// TIA Portal V17 export
// export: Created 2022-03-12T16:05:29.4048686Z, ExportSetting WithDefaults, DisplayName Totally Integrated Automation Portal, DisplayVersion V17, DisplayName TIA Portal Openness, DisplayVersion V17, DisplayName TIA Portal Version Control Interface, DisplayVersion V17, DisplayName STEP 7 Professional, DisplayVersion V17, DisplayName STEP 7 Safety, DisplayVersion V17, DisplayName WinCC Advanced / Unified PC, DisplayVersion V17
DATA_BLOCK "MessagePrefix"   // DB31604
TITLE = CPG_MessagePrefix
{ S7_Optimized_Access := 'TRUE' }
AUTHOR : tech.team.motioncontrol@siemens.com
FAMILY : CPG
VERSION : 1.0
// Support: tech.team.motioncontrol@siemens.com
// Fax: +49 (0) 9131/98-1297
// stored: AutoNumber true, DBAccessibleFromOPCUA true, DBAccessibleFromWebserver true, IsOnlyStoredInLoadMemory false, IsRetainMemResEnabled false, IsWriteProtectedInAS false, MemoryReserve 0
   VAR
      UN { ExternalAccessible := 'False'; ExternalVisible := 'False'; ExternalWritable := 'False'} : Struct   // MessagePrefix for Unit
         Alarm { ExternalAccessible := 'False'; ExternalVisible := 'False'; ExternalWritable := 'False'; S7_SetPoint := 'True'} : "CPG_typeMessagePrefix";   // MessagePrefix for Unit Alarms
      END_STRUCT;
      EM00 { ExternalAccessible := 'False'; ExternalVisible := 'False'; ExternalWritable := 'False'} : Struct   // MessagePrefix for EquipmentModuleEM00
         EventControl { ExternalAccessible := 'False'; ExternalVisible := 'False'; ExternalWritable := 'False'; S7_SetPoint := 'True'} : "CPG_typeMessagePrefix";   // MessagePrefixforEventControl
         CM01 { ExternalAccessible := 'False'; ExternalVisible := 'False'; ExternalWritable := 'False'; S7_SetPoint := 'True'} : "CPG_typeMessagePrefix";   // MessagePrefixforControlModule#01
         CM02 { ExternalAccessible := 'False'; ExternalVisible := 'False'; ExternalWritable := 'False'; S7_SetPoint := 'True'} : "CPG_typeMessagePrefix";   // MessagePrefixforControlModule#02
         CM03 { ExternalAccessible := 'False'; ExternalVisible := 'False'; ExternalWritable := 'False'; S7_SetPoint := 'True'} : "CPG_typeMessagePrefix";   // MessagePrefixforControlModule#03
         CM04 { ExternalAccessible := 'False'; ExternalVisible := 'False'; ExternalWritable := 'False'; S7_SetPoint := 'True'} : "CPG_typeMessagePrefix";   // MessagePrefixforControlModule#04
         CM05 { ExternalAccessible := 'False'; ExternalVisible := 'False'; ExternalWritable := 'False'; S7_SetPoint := 'True'} : "CPG_typeMessagePrefix";   // MessagePrefixforControlModule#05
         CM06 { ExternalAccessible := 'False'; ExternalVisible := 'False'; ExternalWritable := 'False'; S7_SetPoint := 'True'} : "CPG_typeMessagePrefix";   // MessagePrefixforControlModule#06
         CM07 { ExternalAccessible := 'False'; ExternalVisible := 'False'; ExternalWritable := 'False'; S7_SetPoint := 'True'} : "CPG_typeMessagePrefix";   // MessagePrefixforControlModule#07
         CM08 { ExternalAccessible := 'False'; ExternalVisible := 'False'; ExternalWritable := 'False'; S7_SetPoint := 'True'} : "CPG_typeMessagePrefix";   // MessagePrefixforControlModule#08
         CM09 { ExternalAccessible := 'False'; ExternalVisible := 'False'; ExternalWritable := 'False'; S7_SetPoint := 'True'} : "CPG_typeMessagePrefix";   // MessagePrefixforControlModule#09
         CM10 { ExternalAccessible := 'False'; ExternalVisible := 'False'; ExternalWritable := 'False'; S7_SetPoint := 'True'} : "CPG_typeMessagePrefix";   // MessagePrefixforControlModule#10
      END_STRUCT;
      EM01 { ExternalAccessible := 'False'; ExternalVisible := 'False'; ExternalWritable := 'False'} : Struct   // MessagePrefix for EquipmentModuleEM01
         EventControl { ExternalAccessible := 'False'; ExternalVisible := 'False'; ExternalWritable := 'False'; S7_SetPoint := 'True'} : "CPG_typeMessagePrefix";   // MessagePrefixforEventControl
         CM01 { ExternalAccessible := 'False'; ExternalVisible := 'False'; ExternalWritable := 'False'; S7_SetPoint := 'True'} : "CPG_typeMessagePrefix";   // MessagePrefixforControlModule#01
         CM02 { ExternalAccessible := 'False'; ExternalVisible := 'False'; ExternalWritable := 'False'; S7_SetPoint := 'True'} : "CPG_typeMessagePrefix";   // MessagePrefixforControlModule#02
         CM03 { ExternalAccessible := 'False'; ExternalVisible := 'False'; ExternalWritable := 'False'; S7_SetPoint := 'True'} : "CPG_typeMessagePrefix";   // MessagePrefixforControlModule#03
         CM04 { ExternalAccessible := 'False'; ExternalVisible := 'False'; ExternalWritable := 'False'; S7_SetPoint := 'True'} : "CPG_typeMessagePrefix";   // MessagePrefixforControlModule#04
         CM05 { ExternalAccessible := 'False'; ExternalVisible := 'False'; ExternalWritable := 'False'; S7_SetPoint := 'True'} : "CPG_typeMessagePrefix";   // MessagePrefixforControlModule#05
         CM06 { ExternalAccessible := 'False'; ExternalVisible := 'False'; ExternalWritable := 'False'; S7_SetPoint := 'True'} : "CPG_typeMessagePrefix";   // MessagePrefixforControlModule#06
         CM07 { ExternalAccessible := 'False'; ExternalVisible := 'False'; ExternalWritable := 'False'; S7_SetPoint := 'True'} : "CPG_typeMessagePrefix";   // MessagePrefixforControlModule#07
         CM08 { ExternalAccessible := 'False'; ExternalVisible := 'False'; ExternalWritable := 'False'; S7_SetPoint := 'True'} : "CPG_typeMessagePrefix";   // MessagePrefixforControlModule#08
         CM09 { ExternalAccessible := 'False'; ExternalVisible := 'False'; ExternalWritable := 'False'; S7_SetPoint := 'True'} : "CPG_typeMessagePrefix";   // MessagePrefixforControlModule#09
         CM10 { ExternalAccessible := 'False'; ExternalVisible := 'False'; ExternalWritable := 'False'; S7_SetPoint := 'True'} : "CPG_typeMessagePrefix";   // MessagePrefixforControlModule#10
      END_STRUCT;
      EM02 { ExternalAccessible := 'False'; ExternalVisible := 'False'; ExternalWritable := 'False'} : Struct   // MessagePrefix for EquipmentModuleEM02
         EventControl { ExternalAccessible := 'False'; ExternalVisible := 'False'; ExternalWritable := 'False'; S7_SetPoint := 'True'} : "CPG_typeMessagePrefix";   // MessagePrefixforEventControl
         CM01 { ExternalAccessible := 'False'; ExternalVisible := 'False'; ExternalWritable := 'False'; S7_SetPoint := 'True'} : "CPG_typeMessagePrefix";   // MessagePrefixforControlModule#01
         CM02 { ExternalAccessible := 'False'; ExternalVisible := 'False'; ExternalWritable := 'False'; S7_SetPoint := 'True'} : "CPG_typeMessagePrefix";   // MessagePrefixforControlModule#02
         CM03 { ExternalAccessible := 'False'; ExternalVisible := 'False'; ExternalWritable := 'False'; S7_SetPoint := 'True'} : "CPG_typeMessagePrefix";   // MessagePrefixforControlModule#03
         CM04 { ExternalAccessible := 'False'; ExternalVisible := 'False'; ExternalWritable := 'False'; S7_SetPoint := 'True'} : "CPG_typeMessagePrefix";   // MessagePrefixforControlModule#04
         CM05 { ExternalAccessible := 'False'; ExternalVisible := 'False'; ExternalWritable := 'False'; S7_SetPoint := 'True'} : "CPG_typeMessagePrefix";   // MessagePrefixforControlModule#05
         CM06 { ExternalAccessible := 'False'; ExternalVisible := 'False'; ExternalWritable := 'False'; S7_SetPoint := 'True'} : "CPG_typeMessagePrefix";   // MessagePrefixforControlModule#06
         CM07 { ExternalAccessible := 'False'; ExternalVisible := 'False'; ExternalWritable := 'False'; S7_SetPoint := 'True'} : "CPG_typeMessagePrefix";   // MessagePrefixforControlModule#07
         CM08 { ExternalAccessible := 'False'; ExternalVisible := 'False'; ExternalWritable := 'False'; S7_SetPoint := 'True'} : "CPG_typeMessagePrefix";   // MessagePrefixforControlModule#08
         CM09 { ExternalAccessible := 'False'; ExternalVisible := 'False'; ExternalWritable := 'False'; S7_SetPoint := 'True'} : "CPG_typeMessagePrefix";   // MessagePrefixforControlModule#09
         CM10 { ExternalAccessible := 'False'; ExternalVisible := 'False'; ExternalWritable := 'False'; S7_SetPoint := 'True'} : "CPG_typeMessagePrefix";   // MessagePrefixforControlModule#10
      END_STRUCT;
      EM03 { ExternalAccessible := 'False'; ExternalVisible := 'False'; ExternalWritable := 'False'} : Struct   // MessagePrefix for EquipmentModuleEM03
         EventControl { ExternalAccessible := 'False'; ExternalVisible := 'False'; ExternalWritable := 'False'; S7_SetPoint := 'True'} : "CPG_typeMessagePrefix";   // MessagePrefixforEventControl
         CM01 { ExternalAccessible := 'False'; ExternalVisible := 'False'; ExternalWritable := 'False'; S7_SetPoint := 'True'} : "CPG_typeMessagePrefix";   // MessagePrefixforControlModule#01
         CM02 { ExternalAccessible := 'False'; ExternalVisible := 'False'; ExternalWritable := 'False'; S7_SetPoint := 'True'} : "CPG_typeMessagePrefix";   // MessagePrefixforControlModule#02
         CM03 { ExternalAccessible := 'False'; ExternalVisible := 'False'; ExternalWritable := 'False'; S7_SetPoint := 'True'} : "CPG_typeMessagePrefix";   // MessagePrefixforControlModule#03
         CM04 { ExternalAccessible := 'False'; ExternalVisible := 'False'; ExternalWritable := 'False'; S7_SetPoint := 'True'} : "CPG_typeMessagePrefix";   // MessagePrefixforControlModule#04
         CM05 { ExternalAccessible := 'False'; ExternalVisible := 'False'; ExternalWritable := 'False'; S7_SetPoint := 'True'} : "CPG_typeMessagePrefix";   // MessagePrefixforControlModule#05
         CM06 { ExternalAccessible := 'False'; ExternalVisible := 'False'; ExternalWritable := 'False'; S7_SetPoint := 'True'} : "CPG_typeMessagePrefix";   // MessagePrefixforControlModule#06
         CM07 { ExternalAccessible := 'False'; ExternalVisible := 'False'; ExternalWritable := 'False'; S7_SetPoint := 'True'} : "CPG_typeMessagePrefix";   // MessagePrefixforControlModule#07
         CM08 { ExternalAccessible := 'False'; ExternalVisible := 'False'; ExternalWritable := 'False'; S7_SetPoint := 'True'} : "CPG_typeMessagePrefix";   // MessagePrefixforControlModule#08
         CM09 { ExternalAccessible := 'False'; ExternalVisible := 'False'; ExternalWritable := 'False'; S7_SetPoint := 'True'} : "CPG_typeMessagePrefix";   // MessagePrefixforControlModule#09
         CM10 { ExternalAccessible := 'False'; ExternalVisible := 'False'; ExternalWritable := 'False'; S7_SetPoint := 'True'} : "CPG_typeMessagePrefix";   // MessagePrefixforControlModule#10
      END_STRUCT;
      EM04 { ExternalAccessible := 'False'; ExternalVisible := 'False'; ExternalWritable := 'False'} : Struct   // MessagePrefix for EquipmentModuleEM04
         EventControl { ExternalAccessible := 'False'; ExternalVisible := 'False'; ExternalWritable := 'False'; S7_SetPoint := 'True'} : "CPG_typeMessagePrefix";   // MessagePrefixforEventControl
         CM01 { ExternalAccessible := 'False'; ExternalVisible := 'False'; ExternalWritable := 'False'; S7_SetPoint := 'True'} : "CPG_typeMessagePrefix";   // MessagePrefixforControlModule#01
         CM02 { ExternalAccessible := 'False'; ExternalVisible := 'False'; ExternalWritable := 'False'; S7_SetPoint := 'True'} : "CPG_typeMessagePrefix";   // MessagePrefixforControlModule#02
         CM03 { ExternalAccessible := 'False'; ExternalVisible := 'False'; ExternalWritable := 'False'; S7_SetPoint := 'True'} : "CPG_typeMessagePrefix";   // MessagePrefixforControlModule#03
         CM04 { ExternalAccessible := 'False'; ExternalVisible := 'False'; ExternalWritable := 'False'; S7_SetPoint := 'True'} : "CPG_typeMessagePrefix";   // MessagePrefixforControlModule#04
         CM05 { ExternalAccessible := 'False'; ExternalVisible := 'False'; ExternalWritable := 'False'; S7_SetPoint := 'True'} : "CPG_typeMessagePrefix";   // MessagePrefixforControlModule#05
         CM06 { ExternalAccessible := 'False'; ExternalVisible := 'False'; ExternalWritable := 'False'; S7_SetPoint := 'True'} : "CPG_typeMessagePrefix";   // MessagePrefixforControlModule#06
         CM07 { ExternalAccessible := 'False'; ExternalVisible := 'False'; ExternalWritable := 'False'; S7_SetPoint := 'True'} : "CPG_typeMessagePrefix";   // MessagePrefixforControlModule#07
         CM08 { ExternalAccessible := 'False'; ExternalVisible := 'False'; ExternalWritable := 'False'; S7_SetPoint := 'True'} : "CPG_typeMessagePrefix";   // MessagePrefixforControlModule#08
         CM09 { ExternalAccessible := 'False'; ExternalVisible := 'False'; ExternalWritable := 'False'; S7_SetPoint := 'True'} : "CPG_typeMessagePrefix";   // MessagePrefixforControlModule#09
         CM10 { ExternalAccessible := 'False'; ExternalVisible := 'False'; ExternalWritable := 'False'; S7_SetPoint := 'True'} : "CPG_typeMessagePrefix";   // MessagePrefixforControlModule#10
      END_STRUCT;
      EM05 { ExternalAccessible := 'False'; ExternalVisible := 'False'; ExternalWritable := 'False'} : Struct   // MessagePrefix for EquipmentModuleEM05
         EventControl { ExternalAccessible := 'False'; ExternalVisible := 'False'; ExternalWritable := 'False'; S7_SetPoint := 'True'} : "CPG_typeMessagePrefix";   // MessagePrefixforEventControl
         CM01 { ExternalAccessible := 'False'; ExternalVisible := 'False'; ExternalWritable := 'False'; S7_SetPoint := 'True'} : "CPG_typeMessagePrefix";   // MessagePrefixforControlModule#01
         CM02 { ExternalAccessible := 'False'; ExternalVisible := 'False'; ExternalWritable := 'False'; S7_SetPoint := 'True'} : "CPG_typeMessagePrefix";   // MessagePrefixforControlModule#02
         CM03 { ExternalAccessible := 'False'; ExternalVisible := 'False'; ExternalWritable := 'False'; S7_SetPoint := 'True'} : "CPG_typeMessagePrefix";   // MessagePrefixforControlModule#03
         CM04 { ExternalAccessible := 'False'; ExternalVisible := 'False'; ExternalWritable := 'False'; S7_SetPoint := 'True'} : "CPG_typeMessagePrefix";   // MessagePrefixforControlModule#04
         CM05 { ExternalAccessible := 'False'; ExternalVisible := 'False'; ExternalWritable := 'False'; S7_SetPoint := 'True'} : "CPG_typeMessagePrefix";   // MessagePrefixforControlModule#05
         CM06 { ExternalAccessible := 'False'; ExternalVisible := 'False'; ExternalWritable := 'False'; S7_SetPoint := 'True'} : "CPG_typeMessagePrefix";   // MessagePrefixforControlModule#06
         CM07 { ExternalAccessible := 'False'; ExternalVisible := 'False'; ExternalWritable := 'False'; S7_SetPoint := 'True'} : "CPG_typeMessagePrefix";   // MessagePrefixforControlModule#07
         CM08 { ExternalAccessible := 'False'; ExternalVisible := 'False'; ExternalWritable := 'False'; S7_SetPoint := 'True'} : "CPG_typeMessagePrefix";   // MessagePrefixforControlModule#08
         CM09 { ExternalAccessible := 'False'; ExternalVisible := 'False'; ExternalWritable := 'False'; S7_SetPoint := 'True'} : "CPG_typeMessagePrefix";   // MessagePrefixforControlModule#09
         CM10 { ExternalAccessible := 'False'; ExternalVisible := 'False'; ExternalWritable := 'False'; S7_SetPoint := 'True'} : "CPG_typeMessagePrefix";   // MessagePrefixforControlModule#10
      END_STRUCT;
      EM06 { ExternalAccessible := 'False'; ExternalVisible := 'False'; ExternalWritable := 'False'} : Struct   // MessagePrefix for EquipmentModuleEM06
         EventControl { ExternalAccessible := 'False'; ExternalVisible := 'False'; ExternalWritable := 'False'; S7_SetPoint := 'True'} : "CPG_typeMessagePrefix";   // MessagePrefixforEventControl
         CM01 { ExternalAccessible := 'False'; ExternalVisible := 'False'; ExternalWritable := 'False'; S7_SetPoint := 'True'} : "CPG_typeMessagePrefix";   // MessagePrefixforControlModule#01
         CM02 { ExternalAccessible := 'False'; ExternalVisible := 'False'; ExternalWritable := 'False'; S7_SetPoint := 'True'} : "CPG_typeMessagePrefix";   // MessagePrefixforControlModule#02
         CM03 { ExternalAccessible := 'False'; ExternalVisible := 'False'; ExternalWritable := 'False'; S7_SetPoint := 'True'} : "CPG_typeMessagePrefix";   // MessagePrefixforControlModule#03
         CM04 { ExternalAccessible := 'False'; ExternalVisible := 'False'; ExternalWritable := 'False'; S7_SetPoint := 'True'} : "CPG_typeMessagePrefix";   // MessagePrefixforControlModule#04
         CM05 { ExternalAccessible := 'False'; ExternalVisible := 'False'; ExternalWritable := 'False'; S7_SetPoint := 'True'} : "CPG_typeMessagePrefix";   // MessagePrefixforControlModule#05
         CM06 { ExternalAccessible := 'False'; ExternalVisible := 'False'; ExternalWritable := 'False'; S7_SetPoint := 'True'} : "CPG_typeMessagePrefix";   // MessagePrefixforControlModule#06
         CM07 { ExternalAccessible := 'False'; ExternalVisible := 'False'; ExternalWritable := 'False'; S7_SetPoint := 'True'} : "CPG_typeMessagePrefix";   // MessagePrefixforControlModule#07
         CM08 { ExternalAccessible := 'False'; ExternalVisible := 'False'; ExternalWritable := 'False'; S7_SetPoint := 'True'} : "CPG_typeMessagePrefix";   // MessagePrefixforControlModule#08
         CM09 { ExternalAccessible := 'False'; ExternalVisible := 'False'; ExternalWritable := 'False'; S7_SetPoint := 'True'} : "CPG_typeMessagePrefix";   // MessagePrefixforControlModule#09
         CM10 { ExternalAccessible := 'False'; ExternalVisible := 'False'; ExternalWritable := 'False'; S7_SetPoint := 'True'} : "CPG_typeMessagePrefix";   // MessagePrefixforControlModule#10
      END_STRUCT;
      EM07 { ExternalAccessible := 'False'; ExternalVisible := 'False'; ExternalWritable := 'False'} : Struct   // MessagePrefix for EquipmentModuleEM07
         EventControl { ExternalAccessible := 'False'; ExternalVisible := 'False'; ExternalWritable := 'False'; S7_SetPoint := 'True'} : "CPG_typeMessagePrefix";   // MessagePrefixforEventControl
         CM01 { ExternalAccessible := 'False'; ExternalVisible := 'False'; ExternalWritable := 'False'; S7_SetPoint := 'True'} : "CPG_typeMessagePrefix";   // MessagePrefixforControlModule#01
         CM02 { ExternalAccessible := 'False'; ExternalVisible := 'False'; ExternalWritable := 'False'; S7_SetPoint := 'True'} : "CPG_typeMessagePrefix";   // MessagePrefixforControlModule#02
         CM03 { ExternalAccessible := 'False'; ExternalVisible := 'False'; ExternalWritable := 'False'; S7_SetPoint := 'True'} : "CPG_typeMessagePrefix";   // MessagePrefixforControlModule#03
         CM04 { ExternalAccessible := 'False'; ExternalVisible := 'False'; ExternalWritable := 'False'; S7_SetPoint := 'True'} : "CPG_typeMessagePrefix";   // MessagePrefixforControlModule#04
         CM05 { ExternalAccessible := 'False'; ExternalVisible := 'False'; ExternalWritable := 'False'; S7_SetPoint := 'True'} : "CPG_typeMessagePrefix";   // MessagePrefixforControlModule#05
         CM06 { ExternalAccessible := 'False'; ExternalVisible := 'False'; ExternalWritable := 'False'; S7_SetPoint := 'True'} : "CPG_typeMessagePrefix";   // MessagePrefixforControlModule#06
         CM07 { ExternalAccessible := 'False'; ExternalVisible := 'False'; ExternalWritable := 'False'; S7_SetPoint := 'True'} : "CPG_typeMessagePrefix";   // MessagePrefixforControlModule#07
         CM08 { ExternalAccessible := 'False'; ExternalVisible := 'False'; ExternalWritable := 'False'; S7_SetPoint := 'True'} : "CPG_typeMessagePrefix";   // MessagePrefixforControlModule#08
         CM09 { ExternalAccessible := 'False'; ExternalVisible := 'False'; ExternalWritable := 'False'; S7_SetPoint := 'True'} : "CPG_typeMessagePrefix";   // MessagePrefixforControlModule#09
         CM10 { ExternalAccessible := 'False'; ExternalVisible := 'False'; ExternalWritable := 'False'; S7_SetPoint := 'True'} : "CPG_typeMessagePrefix";   // MessagePrefixforControlModule#10
      END_STRUCT;
      EM08 { ExternalAccessible := 'False'; ExternalVisible := 'False'; ExternalWritable := 'False'} : Struct   // MessagePrefix for EquipmentModuleEM08
         EventControl { ExternalAccessible := 'False'; ExternalVisible := 'False'; ExternalWritable := 'False'; S7_SetPoint := 'True'} : "CPG_typeMessagePrefix";   // MessagePrefixforEventControl
         CM01 { ExternalAccessible := 'False'; ExternalVisible := 'False'; ExternalWritable := 'False'; S7_SetPoint := 'True'} : "CPG_typeMessagePrefix";   // MessagePrefixforControlModule#01
         CM02 { ExternalAccessible := 'False'; ExternalVisible := 'False'; ExternalWritable := 'False'; S7_SetPoint := 'True'} : "CPG_typeMessagePrefix";   // MessagePrefixforControlModule#02
         CM03 { ExternalAccessible := 'False'; ExternalVisible := 'False'; ExternalWritable := 'False'; S7_SetPoint := 'True'} : "CPG_typeMessagePrefix";   // MessagePrefixforControlModule#03
         CM04 { ExternalAccessible := 'False'; ExternalVisible := 'False'; ExternalWritable := 'False'; S7_SetPoint := 'True'} : "CPG_typeMessagePrefix";   // MessagePrefixforControlModule#04
         CM05 { ExternalAccessible := 'False'; ExternalVisible := 'False'; ExternalWritable := 'False'; S7_SetPoint := 'True'} : "CPG_typeMessagePrefix";   // MessagePrefixforControlModule#05
         CM06 { ExternalAccessible := 'False'; ExternalVisible := 'False'; ExternalWritable := 'False'; S7_SetPoint := 'True'} : "CPG_typeMessagePrefix";   // MessagePrefixforControlModule#06
         CM07 { ExternalAccessible := 'False'; ExternalVisible := 'False'; ExternalWritable := 'False'; S7_SetPoint := 'True'} : "CPG_typeMessagePrefix";   // MessagePrefixforControlModule#07
         CM08 { ExternalAccessible := 'False'; ExternalVisible := 'False'; ExternalWritable := 'False'; S7_SetPoint := 'True'} : "CPG_typeMessagePrefix";   // MessagePrefixforControlModule#08
         CM09 { ExternalAccessible := 'False'; ExternalVisible := 'False'; ExternalWritable := 'False'; S7_SetPoint := 'True'} : "CPG_typeMessagePrefix";   // MessagePrefixforControlModule#09
         CM10 { ExternalAccessible := 'False'; ExternalVisible := 'False'; ExternalWritable := 'False'; S7_SetPoint := 'True'} : "CPG_typeMessagePrefix";   // MessagePrefixforControlModule#10
      END_STRUCT;
      EM09 { ExternalAccessible := 'False'; ExternalVisible := 'False'; ExternalWritable := 'False'} : Struct   // MessagePrefix for EquipmentModuleEM09
         EventControl { ExternalAccessible := 'False'; ExternalVisible := 'False'; ExternalWritable := 'False'; S7_SetPoint := 'True'} : "CPG_typeMessagePrefix";   // MessagePrefixforEventControl
         CM01 { ExternalAccessible := 'False'; ExternalVisible := 'False'; ExternalWritable := 'False'; S7_SetPoint := 'True'} : "CPG_typeMessagePrefix";   // MessagePrefixforControlModule#01
         CM02 { ExternalAccessible := 'False'; ExternalVisible := 'False'; ExternalWritable := 'False'; S7_SetPoint := 'True'} : "CPG_typeMessagePrefix";   // MessagePrefixforControlModule#02
         CM03 { ExternalAccessible := 'False'; ExternalVisible := 'False'; ExternalWritable := 'False'; S7_SetPoint := 'True'} : "CPG_typeMessagePrefix";   // MessagePrefixforControlModule#03
         CM04 { ExternalAccessible := 'False'; ExternalVisible := 'False'; ExternalWritable := 'False'; S7_SetPoint := 'True'} : "CPG_typeMessagePrefix";   // MessagePrefixforControlModule#04
         CM05 { ExternalAccessible := 'False'; ExternalVisible := 'False'; ExternalWritable := 'False'; S7_SetPoint := 'True'} : "CPG_typeMessagePrefix";   // MessagePrefixforControlModule#05
         CM06 { ExternalAccessible := 'False'; ExternalVisible := 'False'; ExternalWritable := 'False'; S7_SetPoint := 'True'} : "CPG_typeMessagePrefix";   // MessagePrefixforControlModule#06
         CM07 { ExternalAccessible := 'False'; ExternalVisible := 'False'; ExternalWritable := 'False'; S7_SetPoint := 'True'} : "CPG_typeMessagePrefix";   // MessagePrefixforControlModule#07
         CM08 { ExternalAccessible := 'False'; ExternalVisible := 'False'; ExternalWritable := 'False'; S7_SetPoint := 'True'} : "CPG_typeMessagePrefix";   // MessagePrefixforControlModule#08
         CM09 { ExternalAccessible := 'False'; ExternalVisible := 'False'; ExternalWritable := 'False'; S7_SetPoint := 'True'} : "CPG_typeMessagePrefix";   // MessagePrefixforControlModule#09
         CM10 { ExternalAccessible := 'False'; ExternalVisible := 'False'; ExternalWritable := 'False'; S7_SetPoint := 'True'} : "CPG_typeMessagePrefix";   // MessagePrefixforControlModule#10
      END_STRUCT;
   END_VAR
BEGIN
   UN.Alarm.messagePrefix[0..2] := 'Unit ';
   EM00.EventControl.messagePrefix[0..2] := 'EM00 ';
   EM00.CM01.messagePrefix[0..2] := 'CM01 ';
   EM00.CM02.messagePrefix[0..2] := 'CM02 ';
   EM00.CM03.messagePrefix[0..2] := 'CM03 ';
   EM00.CM04.messagePrefix[0..2] := 'CM04 ';
   EM00.CM05.messagePrefix[0..2] := 'CM05 ';
   EM00.CM06.messagePrefix[0..2] := 'CM06 ';
   EM00.CM07.messagePrefix[0..2] := 'CM07 ';
   EM00.CM08.messagePrefix[0..2] := 'CM08 ';
   EM00.CM09.messagePrefix[0..2] := 'CM09 ';
   EM00.CM10.messagePrefix[0..2] := 'CM10 ';
   EM01.EventControl.messagePrefix[0..2] := 'EM01 ';
   EM01.CM01.messagePrefix[0..2] := 'CM01 ';
   EM01.CM02.messagePrefix[0..2] := 'CM02 ';
   EM01.CM03.messagePrefix[0..2] := 'CM03 ';
   EM01.CM04.messagePrefix[0..2] := 'CM04 ';
   EM01.CM05.messagePrefix[0..2] := 'CM05 ';
   EM01.CM06.messagePrefix[0..2] := 'CM06 ';
   EM01.CM07.messagePrefix[0..2] := 'CM07 ';
   EM01.CM08.messagePrefix[0..2] := 'CM08 ';
   EM01.CM09.messagePrefix[0..2] := 'CM09 ';
   EM01.CM10.messagePrefix[0..2] := 'CM10 ';
   EM02.EventControl.messagePrefix[0..2] := 'EM01 ';
   EM02.CM01.messagePrefix[0..2] := 'CM01 ';
   EM02.CM02.messagePrefix[0..2] := 'CM02 ';
   EM02.CM03.messagePrefix[0..2] := 'CM03 ';
   EM02.CM04.messagePrefix[0..2] := 'CM04 ';
   EM02.CM05.messagePrefix[0..2] := 'CM05 ';
   EM02.CM06.messagePrefix[0..2] := 'CM06 ';
   EM02.CM07.messagePrefix[0..2] := 'CM07 ';
   EM02.CM08.messagePrefix[0..2] := 'CM08 ';
   EM02.CM09.messagePrefix[0..2] := 'CM09 ';
   EM02.CM10.messagePrefix[0..2] := 'CM10 ';
   EM03.EventControl.messagePrefix[0..2] := 'EM03 ';
   EM03.CM01.messagePrefix[0..2] := 'CM01 ';
   EM03.CM02.messagePrefix[0..2] := 'CM02 ';
   EM03.CM03.messagePrefix[0..2] := 'CM03 ';
   EM03.CM04.messagePrefix[0..2] := 'CM04 ';
   EM03.CM05.messagePrefix[0..2] := 'CM05 ';
   EM03.CM06.messagePrefix[0..2] := 'CM06 ';
   EM03.CM07.messagePrefix[0..2] := 'CM07 ';
   EM03.CM08.messagePrefix[0..2] := 'CM08 ';
   EM03.CM09.messagePrefix[0..2] := 'CM09 ';
   EM03.CM10.messagePrefix[0..2] := 'CM10 ';
   EM04.EventControl.messagePrefix[0..2] := 'EM04 ';
   EM04.CM01.messagePrefix[0..2] := 'CM01 ';
   EM04.CM02.messagePrefix[0..2] := 'CM02 ';
   EM04.CM03.messagePrefix[0..2] := 'CM03 ';
   EM04.CM04.messagePrefix[0..2] := 'CM04 ';
   EM04.CM05.messagePrefix[0..2] := 'CM05 ';
   EM04.CM06.messagePrefix[0..2] := 'CM06 ';
   EM04.CM07.messagePrefix[0..2] := 'CM07 ';
   EM04.CM08.messagePrefix[0..2] := 'CM08 ';
   EM04.CM09.messagePrefix[0..2] := 'CM09 ';
   EM04.CM10.messagePrefix[0..2] := 'CM10 ';
   EM05.EventControl.messagePrefix[0..2] := 'EM05 ';
   EM05.CM01.messagePrefix[0..2] := 'CM01 ';
   EM05.CM02.messagePrefix[0..2] := 'CM02 ';
   EM05.CM03.messagePrefix[0..2] := 'CM03 ';
   EM05.CM04.messagePrefix[0..2] := 'CM04 ';
   EM05.CM05.messagePrefix[0..2] := 'CM05 ';
   EM05.CM06.messagePrefix[0..2] := 'CM06 ';
   EM05.CM07.messagePrefix[0..2] := 'CM07 ';
   EM05.CM08.messagePrefix[0..2] := 'CM08 ';
   EM05.CM09.messagePrefix[0..2] := 'CM09 ';
   EM05.CM10.messagePrefix[0..2] := 'CM10 ';
   EM06.EventControl.messagePrefix[0..2] := 'EM06 ';
   EM06.CM01.messagePrefix[0..2] := 'CM01 ';
   EM06.CM02.messagePrefix[0..2] := 'CM02 ';
   EM06.CM03.messagePrefix[0..2] := 'CM03 ';
   EM06.CM04.messagePrefix[0..2] := 'CM04 ';
   EM06.CM05.messagePrefix[0..2] := 'CM05 ';
   EM06.CM06.messagePrefix[0..2] := 'CM06 ';
   EM06.CM07.messagePrefix[0..2] := 'CM07 ';
   EM06.CM08.messagePrefix[0..2] := 'CM08 ';
   EM06.CM09.messagePrefix[0..2] := 'CM09 ';
   EM06.CM10.messagePrefix[0..2] := 'CM10 ';
   EM07.EventControl.messagePrefix[0..2] := 'EM07 ';
   EM07.CM01.messagePrefix[0..2] := 'CM01 ';
   EM07.CM02.messagePrefix[0..2] := 'CM02 ';
   EM07.CM03.messagePrefix[0..2] := 'CM03 ';
   EM07.CM04.messagePrefix[0..2] := 'CM04 ';
   EM07.CM05.messagePrefix[0..2] := 'CM05 ';
   EM07.CM06.messagePrefix[0..2] := 'CM06 ';
   EM07.CM07.messagePrefix[0..2] := 'CM07 ';
   EM07.CM08.messagePrefix[0..2] := 'CM08 ';
   EM07.CM09.messagePrefix[0..2] := 'CM09 ';
   EM07.CM10.messagePrefix[0..2] := 'CM10 ';
   EM08.EventControl.messagePrefix[0..2] := 'EM08 ';
   EM08.CM01.messagePrefix[0..2] := 'CM01 ';
   EM08.CM02.messagePrefix[0..2] := 'CM02 ';
   EM08.CM03.messagePrefix[0..2] := 'CM03 ';
   EM08.CM04.messagePrefix[0..2] := 'CM04 ';
   EM08.CM05.messagePrefix[0..2] := 'CM05 ';
   EM08.CM06.messagePrefix[0..2] := 'CM06 ';
   EM08.CM07.messagePrefix[0..2] := 'CM07 ';
   EM08.CM08.messagePrefix[0..2] := 'CM08 ';
   EM08.CM09.messagePrefix[0..2] := 'CM09 ';
   EM08.CM10.messagePrefix[0..2] := 'CM10 ';
   EM09.EventControl.messagePrefix[0..2] := 'EM09 ';
   EM09.CM01.messagePrefix[0..2] := 'CM01 ';
   EM09.CM02.messagePrefix[0..2] := 'CM02 ';
   EM09.CM03.messagePrefix[0..2] := 'CM03 ';
   EM09.CM04.messagePrefix[0..2] := 'CM04 ';
   EM09.CM05.messagePrefix[0..2] := 'CM05 ';
   EM09.CM06.messagePrefix[0..2] := 'CM06 ';
   EM09.CM07.messagePrefix[0..2] := 'CM07 ';
   EM09.CM08.messagePrefix[0..2] := 'CM08 ';
   EM09.CM09.messagePrefix[0..2] := 'CM09 ';
   EM09.CM10.messagePrefix[0..2] := 'CM10 ';
END_DATA_BLOCK
